// TwinCAT 3 PLC project RollingAverageTests
// ProgramVersion: 3.1.4026.22
// libraries:
//   Tc2_Standard, * (Beckhoff Automation GmbH)
//   Tc2_System, * (Beckhoff Automation GmbH)
//   TcUnit, * (www.tcunit.org)
//   B1RollingAverage_Plc,newest,Tc3 Project
// project tree:
//   / PlcTask.TcTTO
//   POUs/ FB_RollingAverageConsumer.TcPOU, MAIN.TcPOU
// (motion and I/O tree: see PLC project b1rollingaverage_plc)

CONFIGURATION RollingAverageTests
    RESOURCE PLC ON TwinCAT3
        TASK PlcTask(INTERVAL := T#10ms, PRIORITY := 21);
        PROGRAM MAIN WITH PlcTask : MAIN;
    END_RESOURCE
END_CONFIGURATION

// ---- POUs/MAIN.TcPOU
PROGRAM MAIN
VAR
END_VAR

END_PROGRAM

// ---- POUs/FB_RollingAverageConsumer.TcPOU
FUNCTION_BLOCK FB_RollingAverageConsumer
VAR
    adder : B1RollingAverage_Plc.FB_RollingAverage;
    lastResult : INT;
END_VAR

lastResult := adder.Step(sample := 10);

END_FUNCTION_BLOCK
